{attribute addProperty BoxType "EL7041-0000-0016"}
{attribute addProperty Id "Latch_C_validBIT10.1251Latch_extern_validBIT10.1252Set_counter_doneBIT10.1253Counter_underflowBIT10.1254Counter_overflowBIT10.1255Extrapolation_stallBIT10.1258Status_of_input_ABIT10.1259Status_of_input_BBIT10.12510Status_of_input_CBIT10.12511Status_of_extern_latchBIT10.12513Sync_errorBIT10.12532TxPDO_ToggleBIT10.1259"}
{attribute addProperty CRC "3603005094"}
{attribute addProperty SizeInBites "16"}
{attribute addProperty SizeInBytes "2"}
TYPE Status_D6C17EA6 :
STRUCT
	{attribute addProperty Name "Latch_C_valid"}
	Latch_C_valid : BIT;
	{attribute addProperty Name "Latch_extern_valid"}
	Latch_extern_valid : BIT;
	{attribute addProperty Name "Set_counter_done"}
	Set_counter_done : BIT;
	{attribute addProperty Name "Counter_underflow"}
	Counter_underflow : BIT;
	{attribute addProperty Name "Counter_overflow"}
	Counter_overflow : BIT;
	{attribute 'hide'}
	reserve_1_BIT_0 : BIT;
	{attribute 'hide'}
	reserve_1_BIT_1 : BIT;
	{attribute addProperty Name "Extrapolation_stall"}
	Extrapolation_stall : BIT;
	{attribute addProperty Name "Status_of_input_A"}
	Status_of_input_A : BIT;
	{attribute addProperty Name "Status_of_input_B"}
	Status_of_input_B : BIT;
	{attribute addProperty Name "Status_of_input_C"}
	Status_of_input_C : BIT;
	{attribute 'hide'}
	reserve_2 : BIT;
	{attribute addProperty Name "Status_of_extern_latch"}
	Status_of_extern_latch : BIT;
	{attribute addProperty Name "Sync_error"}
	Sync_error : BIT;
	{attribute 'hide'}
	reserve_3 : BIT;
	{attribute addProperty Name "TxPDO_Toggle"}
	TxPDO_Toggle : BIT;
END_STRUCT
END_TYPE

(* stored: Version 1.2.0.0, ProductVersion 3.1.4024.9
   DUT Status_D6C17EA6: Id {b3f6b9d9-fd7b-4339-b517-c1a35e2dcfc6} *)
